// TIA Portal V20 export
TYPE "typeCmControlNodeInterlock"
// stored: Namespace Unit1.Em13
   STRUCT
      jrUnIoadingPnPAxisX : "LER_typeAxisInterlock";
      jrUnIoadingPnPAxisZ : "LER_typeAxisInterlock";
      jrUnIoadingPnPAxisC : "LER_typeAxisInterlock";
      jrUnIoadingPnPClamp : "LER_typeTwoWayActuatorInterlock";
   END_STRUCT;
END_TYPE
